Fanuc KAREL source: ko00004.KL

-- PROVISIONAL review KL for V770-1; original PC SHA256 feaef87a0414a81d0437e055504b8ddb08970986ae357d14c50f5194d99e87d4
-- Incomplete behavior may be omitted. Consult companion uncertainty JSON. Do not deploy.
PROGRAM KO00004
%NOLOCKGROUP
-- UNRESOLVED_DECL P1 type=000101
-- UNRESOLVED_DECL P2 type=000101
-- UNRESOLVED_DECL P3 type=000101
-- UNRESOLVED_DECL OUT type=000199
BEGIN
  -- UNRESOLVED_PC offsets 5-56; opcodes 27,22,1C,22,1C,22,1C,76,7E,4A
  -- UNRESOLVED_PC offsets 61-65; opcodes 7F
END KO00004
